{attribute 'qualified_only'}
{attribute 'strict'}
TYPE 
	MachineSubTypeEnum				: (None, CE);
END_TYPE

(* stored: Version 1.1.0.1, ProductVersion 3.1.4024.9
   DUT MachineSubTypeEnum: Id {42385dae-3144-4cc8-a41f-b0fd8482ec3c} *)
